// TwinCAT 3 PLC project test1
// ProgramVersion: 3.1.4026.22
// libraries:
//   Tc2_Standard, * (Beckhoff Automation GmbH)
//   Tc2_System, * (Beckhoff Automation GmbH)
// project tree:
//   GVLs/ SPS.TcGVL
//   / PlcTask.TcTTO
//   POUs/ FB_MeinFunktionsbaustein.TcPOU, MAIN.TcPOU
// real-time tasks:
//   TASK PlcTask: cycle T#10ms, priority 6, ADS port 350
// I/O:
//   DEVICE Gerät 1 (EtherCAT), AmsNetId 5.176.211.3.2.1
//     Klemme 1 (EK1200) [EK1200-7000 EtherCAT Netzteil (1,5A E-Bus)]
//       Klemme 2 (EL1809) [EL1809 16K. Dig. Eingang 24V, 3ms]
//       Klemme 3 (EL9011) [EL9011 Endklemme]
//   DEVICE Gerät 2 (NOV-DP-RAM)
//   DEVICE Gerät 3 (Onboard I/O Device), AmsNetId 5.176.211.3.4.1
//     Klemme 1 (CX7028) [CX7028-0000-0121]
//       modules: Module 1 (DIO_2x), Module 2 (Empty Module), Module 3 (DIO_2x), Module 4 (Empty Module), Module 5 (DI_2x), Module 6 (Empty Module), Module 7 (DI_2x), Module 8 (Empty Module)
//   DEVICE Gerät 4 (CX7050), AmsNetId 5.176.211.3.5.1
// variable links:
//   Device 3 (Onboard I/O Device) <-> Device 1 (EtherCAT)/Term 1 (EK1200)/Term 2 (EL1809)
//     Outputs/Ctrl <-> InfoData/State
//   test1/test1 Instance <-> Device 1 (EtherCAT)/Term 1 (EK1200)/Term 2 (EL1809)
//     PlcTask Inputs/MAIN.fb_MeinFunktionsbaustein.iMeinSensor1 <-> Channel 1/=CPU01+SPS01-B01
//     PlcTask Inputs/SPS.B103 <-> Channel 3/Input 3 ADR26.2

CONFIGURATION test1
    RESOURCE PLC ON TwinCAT3
        TASK PlcTask(INTERVAL := T#10ms, PRIORITY := 6);
        PROGRAM MAIN WITH PlcTask : MAIN;
    END_RESOURCE
END_CONFIGURATION

// ---- GVLs/SPS.TcGVL
{attribute 'qualified_only'}
VAR_GLOBAL
	B103 AT %I* : BOOL; // Füllstand 1
	B104 AT %I* : BOOL; // Füllstand 2
	B105 AT %I* : BOOL; // Füllstand 2
	B106 AT %I* : BOOL; // Füllstand 2
END_VAR

// ---- POUs/MAIN.TcPOU
PROGRAM MAIN
VAR
	bRunOnlyOnce : bool := FALSE;
	msgCtrMask: INT;
	strArg: STRING;
	bInputSensorB01: BOOL;
	fb_MeinFunktionsbaustein : FB_MeinFunktionsbaustein;
	
END_VAR

fb_MeinFunktionsbaustein();

IF NOT bRunOnlyOnce THEN 
	ADSLOGSTR(msgCtrlMask := ADSLOG_MSGTYPE_ERROR OR ADSLOG_MSGTYPE_LOG,
		msgFmtStr := 'Hello World my new',
		strArg := '');
		bRunOnlyOnce := FALSE;
		bInputSensorB01 := TRUE;
		
END_IF

END_PROGRAM

// ---- POUs/FB_MeinFunktionsbaustein.TcPOU
FUNCTION_BLOCK FB_MeinFunktionsbaustein
VAR_INPUT
	iMeinSensor1 AT %I* : BOOL;
	iMeinSensor2 AT %I* : BOOL;
 
END_VAR

iMeinSensor1 := TRUE;
iMeinSensor2 := TRUE;

END_FUNCTION_BLOCK
